PROGRAM MAIN
VAR
   _sampleContext : SampleContext;
END_VAR

_sampleContext.Run();

END_PROGRAM

(* stored: Version 1.1.0.1, ProductVersion 3.1.4024.9
   POU MAIN: Id {d9bafd5f-9ffe-01a0-23ed-be6793c9dbf6}, SpecialFunc None *)
